(* PLC project CoDeSys External Library Template, WAGO e!COCKPIT e!COCKPIT, author 3S - Smart Software Solutions GmbH *)
(* stored: creationDateTime 2019-10-29T12:22:40.817377, version 3.5.5.30, modificationDateTime 2019-10-24T14:40:07.960949, organization 3S - Smart Software Solutions GmbH *)
(* Library project template with all possible element types, docu and a sample project structure *)

FUNCTION fnIDOdbiorcyMatch : BOOL
  VAR_INPUT
    sKomunikat : alSTRINGKomunikat;
    sIDObiektu : STRING;
  END_VAR
  VAR
    typKomunikat : typKomunikat;
    intPetla : INT;
    xMatch : BOOL := TRUE;
    intBlad : INT;
  END_VAR

            fnKomunikatInOut(	xStringNaStrukture := TRUE ,
					xStringUpdateZeStruktury := FALSE ,
					xStrukturyNaString := FALSE ,
					xWyczyscStrukture := FALSE ,
					xAktualizujZnacznikCzasu := FALSE ,
					xAktualizujDlugoscDanych := FALSE ,
					sKomunikat := sKomunikat ,
					typKomunikat := typKomunikat ,
					intBlad := intBlad);

FOR intPetla := 1 TO LEN(sIDObiektu) BY 1 DO
	IF (MID(typKomunikat.sIDPrzeznaczenia , 1 , intPetla) <> MID(sIDObiektu,1,intPetla)) AND MID(typKomunikat.sIDPrzeznaczenia , 1 , intPetla) <> '*' THEN
		xMatch := FALSE;
		EXIT;
	END_IF
END_FOR
fnIDOdbiorcyMatch := xMatch;
          
END_FUNCTION
